FUNCTION_BLOCK TcoRemoteTaskTest EXTENDS TcoCore.TcoObject
VAR
	_invokeInitializedCSharpMethod : TcoCore.TcoRemoteTask(THIS^, NO.Structure);
    _invokeNotInitializedCSharpMethod : TcoCore.TcoRemoteTask(THIS^, NO.Structure);
    _exceptionInMethodWillResultInException : TcoCore.TcoRemoteTask(THIS^, NO.Structure);
END_VAR

_invokeInitializedCSharpMethod();
_invokeNotInitializedCSharpMethod();
_exceptionInMethodWillResultInException();

END_FUNCTION_BLOCK

(* stored: Version 1.1.0.1
   POU TcoRemoteTaskTest: Id {8b2e52e7-ca9d-013a-11b6-88a18f8a3d16}, SpecialFunc None *)
